FUNCTION F_PressAtVacSP : BOOL
VAR_INPUT
END_VAR
VAR
END_VAR

F_PressAtVacSP := //DREAM_NC_GCC_01.IG.rPRESS < ATVAC_INTERLOCK_SP AND DREAM_NC_GCC_01.IG.xPRESS_OK AND
                  //DREAM_DP1_GHC_01.IG.rPRESS < ATVAC_INTERLOCK_SP AND DREAM_DP1_GHC_01.IG.xPRESS_OK AND
                  //DREAM_DP2_GHC_01.IG.rPRESS < ATVAC_INTERLOCK_SP AND DREAM_DP2_GHC_01.IG.xPRESS_OK AND
                  //DREAM_DP3_GHC_01.IG.rPRESS < ATVAC_INTERLOCK_SP AND DREAM_DP3_GHC_01.IG.xPRESS_OK AND
                  //DREAM_CAT1_GHC_01.IG.rPRESS < ATVAC_INTERLOCK_SP AND DREAM_CAT1_GHC_01.IG.xPRESS_OK AND
                  //DREAM_CAT2_GHC_01.IG.rPRESS < ATVAC_INTERLOCK_SP AND DREAM_CAT2_GHC_01.IG.xPRESS_OK AND
                  GVL_VAC_GAUGES.stDREAM_MC_GAUGE.rPRESS < AT_VAC_SP AND GVL_VAC_GAUGES.stDREAM_MC_GAUGE.xPRESS_OK;
                  //GVL_VAC_GAUGES.stDREAM_MC_GHC.xAT_VAC;
                  //we could also be checking ST_VG.xAT_VAC flag and make this value changeable?

END_FUNCTION

(* stored: Version 1.1.0.1, ProductVersion 3.1.4024.12
   POU F_PressAtVacSP: Id {d799ff72-808d-4ce9-b24c-7aac3b16009f}, SpecialFunc None *)
